// TIA Portal V17 export
// export: Created 2025-03-07T09:24:10.9679489Z, ExportSetting WithDefaults, DisplayName Totally Integrated Automation Portal, DisplayVersion V17 Update 8, DisplayName TIA Portal Openness, DisplayVersion V17 Update 8, DisplayName TIA Portal Version Control Interface, DisplayVersion V17, DisplayName SINAMICS Startdrive Advanced, DisplayVersion V17 SP2, DisplayName SINAMICS Startdrive G110M, G120, G120C, G120D, G120P, G115D, DisplayVersion V17 SP2, DisplayName SINAMICS Startdrive G130, G150, S120, S150, SINAMICS MV, S210, DisplayVersion V17 SP2, DisplayName STEP 7 Professional, DisplayVersion V17 Update 8, DisplayName SINUMERIK ONE STEP 7 Toolbox, DisplayVersion V17 Update 12, DisplayName SINUMERIK 840D sl STEP 7 Toolbox, DisplayVersion V17 Update 12, DisplayName STEP 7 Safety, DisplayVersion V17 Update 6, DisplayName WinCC Advanced, DisplayVersion V17 Update 8
DATA_BLOCK "DB22103_POWDER_FLOW_HOPPER_1_UNIT_01"   // DB22103
{ DB_Accessible_From_OPC_UA := 'FALSE' }
VERSION : 0.1
// stored: AutoNumber false, DBAccessibleFromOPCUA false, DBAccessibleFromWebserver true, InstanceOfName FB22102_POWDER_FLOW_SENSOR, InstanceOfType FB
"FB22102_POWDER_FLOW_SENSOR"
   // VAR_INPUT
   //    iANALOG_INPUT : UInt;
   // END_VAR
   // VAR_OUTPUT
   //    oPOWDER_FLOW_ON : Bool;
   //    oWARNING_LIMIT : Bool;
   // END_VAR
   // VAR RETAIN
   //    OUTPUT : Struct
   //       VALUE : Real;
   //    END_STRUCT;
   //    INPUT_SETTINGS : Struct
   //       LOW_RANGE : Real;
   //       HIGH_RANGE : Real;
   //       LOW_LIM_TO_FLOW_ON : Real;
   //       UNIT_NUMBER : Int := 1;
   //       HOPPER_NUMBER : Int := 1;
   //    END_STRUCT;
   //    ALARM_SETTINGS : Struct
   //       WARN_LIMIT_LOW : Real;
   //       WARN_LIMIT_HIGH : Real;
   //       ERROR_CONFIGURATION : Bool;
   //    END_STRUCT;
   //    LOG : Struct
   //       SPARE : Bool;
   //    END_STRUCT;
   // END_VAR
BEGIN
END_DATA_BLOCK
